{attribute 'GeneratedUsingTerminal: KL2761'}
{attribute addProperty BoxType "KL2761"}
{attribute addProperty Id "Channel_1AT %Q*Channel_6576A6810"}
{attribute addProperty CRC "1632160004"}
{attribute addProperty Size "0"}
TYPE KL2761_6148C904 :
STRUCT
	{attribute addProperty Name "Channel_1"}
	Channel_1 : Channel_6576A681;
END_STRUCT
END_TYPE

(* stored: Version 1.2.0.0, ProductVersion 3.1.4024.9
   DUT KL2761_6148C904: Id {768e4c67-e501-4a4b-8317-feefc0010c23} *)
